{attribute addProperty BoxType "EM7004-0000-9995"}
{attribute addProperty Id "OutputAT %Q*ARRAY[0 ..15] OF BOOL128160"}
{attribute addProperty CRC "1232143113"}
{attribute addProperty SizeInBites "128"}
{attribute addProperty SizeInBytes "16"}
TYPE Digital_BF554446 :
STRUCT
	{attribute addProperty Name "Output"}
	Output AT %Q* : ARRAY[0 ..15] OF BOOL;
END_STRUCT
END_TYPE

(* stored: Version 1.2.0.0, ProductVersion 3.1.4024.9
   DUT Digital_BF554446: Id {61b36166-e4dc-4302-acd8-1134d5a7e5d8} *)
